PROGRAM MAIN
VAR
END_VAR

task31();
caseTest();

END_PROGRAM

(* stored: Version 1.1.0.1, ProductVersion 3.1.4024.12
   POU MAIN: Id {5ae94e95-72f5-44cb-9013-79c0156b576e}, SpecialFunc None *)
